# EPICS substitutions: iocBoot/iocvirPV/DPU03.substitutions
file "../../db/virAi.template"{ pattern
{DPU,    num,    Temp}
{03,    0,    500}
{03,    1,    500}
{03,    2,    500}
{03,    3,    500}
{03,    4,    500}
{03,    5,    500}
{03,    6,    500}
{03,    7,    500}
{03,    8,    500}
{03,    9,    500}
{03,    10,    500}
{03,    11,    500}
{03,    12,    500}
{03,    13,    500}
{03,    14,    500}
{03,    15,    500}
{03,    16,    500}
{03,    17,    500}
{03,    18,    500}
{03,    19,    500}
{03,    20,    500}
{03,    21,    500}
{03,    22,    500}
{03,    23,    500}
{03,    24,    500}
{03,    25,    500}
{03,    26,    500}
{03,    27,    500}
{03,    28,    500}
{03,    29,    500}
{03,    30,    500}
{03,    31,    500}
{03,    32,    500}
{03,    33,    500}
{03,    34,    500}
{03,    35,    500}
{03,    36,    500}
{03,    37,    500}
{03,    38,    500}
{03,    39,    500}
{03,    40,    500}
{03,    41,    500}
{03,    42,    500}
{03,    43,    500}
{03,    44,    500}
{03,    45,    500}
{03,    46,    500}
{03,    47,    500}
{03,    48,    500}
{03,    49,    500}
{03,    50,    500}
{03,    51,    500}
{03,    52,    500}
{03,    53,    500}
{03,    54,    500}
{03,    55,    500}
{03,    56,    500}
{03,    57,    500}
{03,    58,    500}
{03,    59,    500}
{03,    60,    500}
{03,    61,    500}
{03,    62,    500}
{03,    63,    500}
{03,    64,    500}
{03,    65,    500}
{03,    66,    500}
{03,    67,    500}
{03,    68,    500}
{03,    69,    500}
{03,    70,    500}
{03,    71,    500}
{03,    72,    500}
{03,    73,    500}
{03,    74,    500}
{03,    75,    500}
{03,    76,    500}
{03,    77,    500}
{03,    78,    500}
{03,    79,    500}
{03,    80,    500}
{03,    81,    500}
{03,    82,    500}
{03,    83,    500}
{03,    84,    500}
{03,    85,    500}
{03,    86,    500}
{03,    87,    500}
{03,    88,    500}
{03,    89,    500}
{03,    90,    500}
{03,    91,    500}
{03,    92,    500}
{03,    93,    500}
{03,    94,    500}
{03,    95,    500}
{03,    96,    500}
{03,    97,    500}
{03,    98,    500}
{03,    99,    500}
{03,    100,    500}
{03,    101,    500}
{03,    102,    500}
{03,    103,    500}
{03,    104,    500}
{03,    105,    500}
{03,    106,    500}
{03,    107,    500}
{03,    108,    500}
{03,    109,    500}
{03,    110,    500}
{03,    111,    500}
{03,    112,    500}
{03,    113,    500}
{03,    114,    500}
{03,    115,    500}
{03,    116,    500}
{03,    117,    500}
{03,    118,    500}
{03,    119,    500}
{03,    120,    500}
{03,    121,    500}
{03,    122,    500}
{03,    123,    500}
{03,    124,    500}
{03,    125,    500}
{03,    126,    500}
{03,    127,    500}
{03,    128,    500}
{03,    129,    500}
{03,    130,    500}
{03,    131,    500}
{03,    132,    500}
{03,    133,    500}
{03,    134,    500}
{03,    135,    500}
{03,    136,    500}
{03,    137,    500}
{03,    138,    500}
{03,    139,    500}
{03,    140,    500}
{03,    141,    500}
{03,    142,    500}
{03,    143,    500}
{03,    144,    500}
{03,    145,    500}
{03,    146,    500}
{03,    147,    500}
{03,    148,    500}
{03,    149,    500}
{03,    150,    500}
{03,    151,    500}
{03,    152,    500}
{03,    153,    500}
{03,    154,    500}
{03,    155,    500}
{03,    156,    500}
{03,    157,    500}
{03,    158,    500}
{03,    159,    500}
{03,    160,    500}
{03,    161,    500}
{03,    162,    500}
{03,    163,    500}
{03,    164,    500}
{03,    165,    500}
{03,    166,    500}
{03,    167,    500}
{03,    168,    500}
{03,    169,    500}
{03,    170,    500}
{03,    171,    500}
{03,    172,    500}
{03,    173,    500}
{03,    174,    500}
{03,    175,    500}
{03,    176,    500}
{03,    177,    500}
{03,    178,    500}
{03,    179,    500}
{03,    180,    500}
{03,    181,    500}
{03,    182,    500}
{03,    183,    500}
{03,    184,    500}
{03,    185,    500}
{03,    186,    500}
{03,    187,    500}
{03,    188,    500}
{03,    189,    500}
{03,    190,    500}
{03,    191,    500}
{03,    192,    500}
{03,    193,    500}
{03,    194,    500}
{03,    195,    500}
{03,    196,    500}
{03,    197,    500}
{03,    198,    500}
{03,    199,    500}
}
